// LS Electric XG5000 project: fda
// PLC LSPLC
// module base 0 slot 0: 입출력 모듈:XBC-DR32H (DC 24V 입력, 릴레이 출력 32점)
// module base 0 slot 1: 위치결정 모듈:XBF-PD02A (위치결정 펄스(LD)출력형, 2축)
// module base 0 slot 2: 출력 모듈:XBE-TN/TP16A (트랜지스터 출력, 16점 (싱크출력/소스출력))

PROGRAM NewProgram (task: 스캔 프로그램)

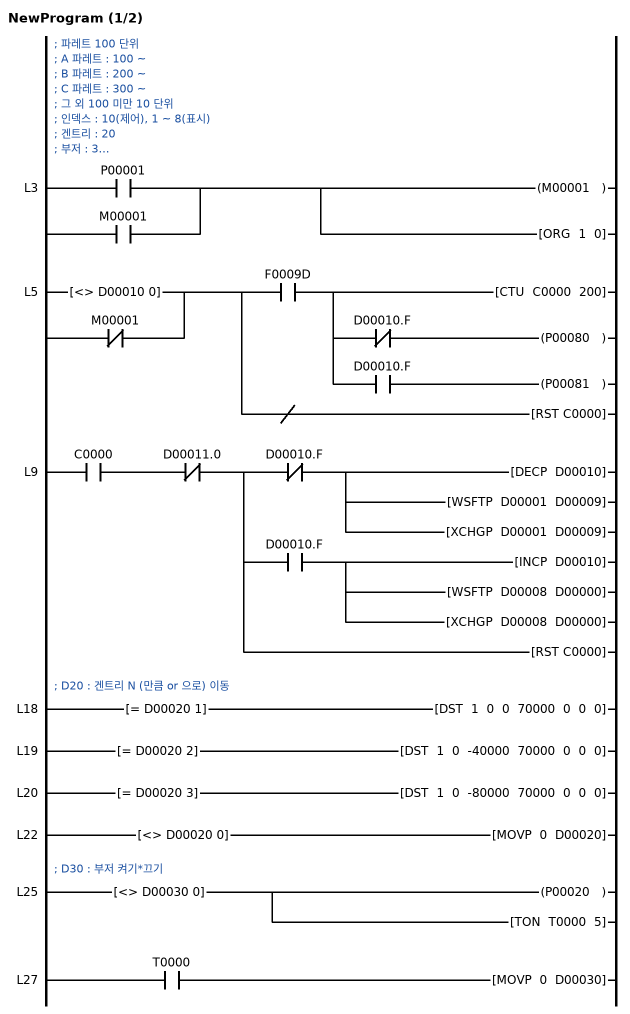
// 파레트 100 단위
// A 파레트 : 100 ~
// B 파레트 : 200 ~
// C 파레트 : 300 ~
// 
// 그 외 100 미만 10 단위
// 인덱스 : 10(제어), 1 ~ 8(표시)
// 겐트리 : 20
// 부저 : 30
// 공압 : 40
// D10 : 인덱스
; L3
LOAD      P00001
OR        M00001
OUT       M00001
ORG       1 0
; L5
LOAD<>    D00010 0
OR NOT    M00001
MPUSH
AND       F0009D
CTU       C0000 200
MPUSH
AND NOT   D00010.F
OUT       P00080
MPOP
AND       D00010.F
OUT       P00081
MPOP
NOT
RST       C0000
; L9
LOAD      C0000
AND NOT   D00011.0
MPUSH
AND NOT   D00010.F
DECP      D00010
WSFTP     D00001 D00009
XCHGP     D00001 D00009
MLOAD
AND       D00010.F
INCP      D00010
WSFTP     D00008 D00000
XCHGP     D00008 D00000
MPOP
RST       C0000
// D20 : 겐트리 N (만큼 or 으로) 이동 
; L18
LOAD=     D00020 1
DST       1 0 0 70000 0 0 0
; L19
LOAD=     D00020 2
DST       1 0 -40000 70000 0 0 0
; L20
LOAD=     D00020 3
DST       1 0 -80000 70000 0 0 0
; L22
LOAD<>    D00020 0
MOVP      0 D00020
// D30 : 부저 켜기*끄기
; L25
LOAD<>    D00030 0
OUT       P00020
TON       T0000 5
; L27
LOAD      T0000
MOVP      0 D00030

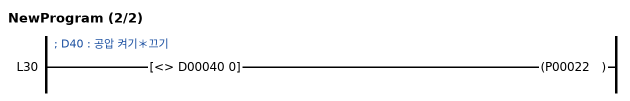
// D40 : 공압 켜기＊끄기
; L30
LOAD<>    D00040 0
OUT       P00022